    CFF_RETURN_LOCAL:
        IF NOT bReturnEntryBlocked THEN
            IF bReturnPublicationAllowed THEN
                IF bStateEntry THEN
                    udiZCommandId := udiZCommandId + 1;
                    IF udiZCommandId = 0 THEN
                        udiZCommandId := 1;
                    END_IF
                END_IF
                stMotionIntent.stZCommand.bEnable := TRUE;
                stMotionIntent.stZCommand.bReset := FALSE;
                stMotionIntent.stZCommand.bStop := FALSE;
                stMotionIntent.stZCommand.bHome := FALSE;
                stMotionIntent.stZCommand.bMoveAbsolute := TRUE;
                stMotionIntent.stZCommand.bMoveVelocity := FALSE;
                stMotionIntent.stZCommand.bUseExternalSetpoint := FALSE;
                stMotionIntent.stZCommand.rHomePosition_mm := 0.0;
                stMotionIntent.stZCommand.rPosition_mm := rCycleStartZPosition_mm;
                stMotionIntent.stZCommand.rVelocity_mm_s :=
                    stCycleSnapshot.stProgram.stHeader.fReturnVelocityMmS;
                stMotionIntent.stZCommand.rAcceleration_mm_s2 :=
                    stSequenceConfigSnapshot.fStandardMoveAccelerationMmS2;
                stMotionIntent.stZCommand.rDeceleration_mm_s2 :=
                    stSequenceConfigSnapshot.fStandardMoveDecelerationMmS2;
                stMotionIntent.stZCommand.eOwnerRequest := Z_OWNER_RETRACT;
                stMotionIntent.bExternalEnableRequest := FALSE;
                stMotionIntent.bExternalDisableRequest := FALSE;
                stMotionIntent.rExternalTargetVelocity_mm_s := 0.0;
                stMotionIntent.bForceProcessExitComplete := TRUE;
                stMotionIntent.bRAxisProcessRequested := TRUE;
                stMotionIntent.stRCommand.bEnable := TRUE;
                stMotionIntent.stRCommand.bReset := FALSE;
                stMotionIntent.stRCommand.bStop := TRUE;
                stMotionIntent.stRCommand.bMoveVelocity := FALSE;
                stMotionIntent.stRCommand.rVelocity_rpm := 0.0;
                stMotionIntent.stRCommand.rAcceleration_rpm_s :=
                    stRAxisProfileSnapshot.fSpeedRampRpmS;
                stMotionIntent.stRCommand.rDeceleration_rpm_s :=
                    stRAxisProfileSnapshot.fSpeedRampRpmS;
                bForceControlEnable := FALSE;
                IF tonReturn.Q THEN
                    IF udiFirstFaultId = 0 THEN
                        udiFirstFaultId := 16#0000A015;
                    END_IF
                    eExitIntent := CFF_EXIT_FAULT_NO_RETURN;
                    eNextState := CFF_FAULT;
                END_IF
                IF (GVL_Status.stFast.udiAcceptedSequenceZCommandId = udiZCommandId)
                    AND GVL_Status.stFast.stZAxis.bDone
                    AND GVL_Status.stFast.stZAxis.bStandstill
                    AND NOT tonReturn.Q THEN
                    eNextState := CFF_EVALUATE;
                END_IF
            ELSE
                IF udiFirstFaultId = 0 THEN
                    udiFirstFaultId := 16#0000A016;
                END_IF
                eExitIntent := CFF_EXIT_FAULT_NO_RETURN;
                eNextState := CFF_FAULT;
            END_IF
        END_IF
    CFF_RETURN_REFERENCE:
        IF NOT bReturnEntryBlocked THEN
            IF bReturnPublicationAllowed THEN
                IF bStateEntry THEN
                    udiZCommandId := udiZCommandId + 1;
                    IF udiZCommandId = 0 THEN
                        udiZCommandId := 1;
                    END_IF
                END_IF
                stMotionIntent.stZCommand.bEnable := TRUE;
                stMotionIntent.stZCommand.bReset := FALSE;
                stMotionIntent.stZCommand.bStop := FALSE;
                stMotionIntent.stZCommand.bHome := FALSE;
                stMotionIntent.stZCommand.bMoveAbsolute := TRUE;
                stMotionIntent.stZCommand.bMoveVelocity := FALSE;
                stMotionIntent.stZCommand.bUseExternalSetpoint := FALSE;
                stMotionIntent.stZCommand.rHomePosition_mm := 0.0;
                stMotionIntent.stZCommand.rPosition_mm :=
                    stCycleSnapshot.stProgram.stHeader.fReturnOpeningMm;
                stMotionIntent.stZCommand.rVelocity_mm_s :=
                    stCycleSnapshot.stProgram.stHeader.fReturnVelocityMmS;
                stMotionIntent.stZCommand.rAcceleration_mm_s2 :=
                    stSequenceConfigSnapshot.fStandardMoveAccelerationMmS2;
                stMotionIntent.stZCommand.rDeceleration_mm_s2 :=
                    stSequenceConfigSnapshot.fStandardMoveDecelerationMmS2;
                stMotionIntent.stZCommand.eOwnerRequest := Z_OWNER_RETRACT;
                stMotionIntent.bExternalEnableRequest := FALSE;
                stMotionIntent.bExternalDisableRequest := FALSE;
                stMotionIntent.rExternalTargetVelocity_mm_s := 0.0;
                stMotionIntent.bForceProcessExitComplete := TRUE;
                stMotionIntent.bRAxisProcessRequested := TRUE;
                stMotionIntent.stRCommand.bEnable := TRUE;
                stMotionIntent.stRCommand.bReset := FALSE;
                stMotionIntent.stRCommand.bStop := TRUE;
                stMotionIntent.stRCommand.bMoveVelocity := FALSE;
                stMotionIntent.stRCommand.rVelocity_rpm := 0.0;
                stMotionIntent.stRCommand.rAcceleration_rpm_s :=
                    stRAxisProfileSnapshot.fSpeedRampRpmS;
                stMotionIntent.stRCommand.rDeceleration_rpm_s :=
                    stRAxisProfileSnapshot.fSpeedRampRpmS;
                bForceControlEnable := FALSE;
                IF tonReturn.Q THEN
                    IF udiFirstFaultId = 0 THEN
                        udiFirstFaultId := 16#0000A015;
                    END_IF
                    eExitIntent := CFF_EXIT_FAULT_NO_RETURN;
                    eNextState := CFF_FAULT;
                END_IF
                IF (GVL_Status.stFast.udiAcceptedSequenceZCommandId = udiZCommandId)
                    AND GVL_Status.stFast.stZAxis.bDone
                    AND GVL_Status.stFast.stZAxis.bStandstill
                    AND NOT tonReturn.Q THEN
                    eNextState := CFF_EVALUATE;
                END_IF
            ELSE
                IF udiFirstFaultId = 0 THEN
                    udiFirstFaultId := 16#0000A016;
                END_IF
                eExitIntent := CFF_EXIT_FAULT_NO_RETURN;
                eNextState := CFF_FAULT;
            END_IF
        END_IF
    CFF_EVALUATE:
        stMotionIntent.stZCommand.bEnable := TRUE;
        stMotionIntent.stZCommand.bReset := FALSE;
        stMotionIntent.stZCommand.bStop := FALSE;
        stMotionIntent.stZCommand.bHome := FALSE;
        stMotionIntent.stZCommand.bMoveAbsolute := TRUE;
        stMotionIntent.stZCommand.bMoveVelocity := FALSE;
        stMotionIntent.stZCommand.bUseExternalSetpoint := FALSE;
        stMotionIntent.stZCommand.rHomePosition_mm := 0.0;
        stMotionIntent.stZCommand.rPosition_mm := SEL(
            stCycleSnapshot.stProgram.stHeader.eReturnMode = RETURN_MODE_REFERENCE,
            rCycleStartZPosition_mm,
            stCycleSnapshot.stProgram.stHeader.fReturnOpeningMm);
        stMotionIntent.stZCommand.rVelocity_mm_s :=
            stCycleSnapshot.stProgram.stHeader.fReturnVelocityMmS;
        stMotionIntent.stZCommand.rAcceleration_mm_s2 :=
            stSequenceConfigSnapshot.fStandardMoveAccelerationMmS2;
        stMotionIntent.stZCommand.rDeceleration_mm_s2 :=
            stSequenceConfigSnapshot.fStandardMoveDecelerationMmS2;
        stMotionIntent.stZCommand.eOwnerRequest := Z_OWNER_RETRACT;
        stMotionIntent.bExternalEnableRequest := FALSE;
        stMotionIntent.bExternalDisableRequest := FALSE;
        stMotionIntent.rExternalTargetVelocity_mm_s := 0.0;
        stMotionIntent.bForceProcessExitComplete := TRUE;
        stMotionIntent.bRAxisProcessRequested := TRUE;
        stMotionIntent.stRCommand.bEnable := TRUE;
        stMotionIntent.stRCommand.bReset := FALSE;
        stMotionIntent.stRCommand.bStop := TRUE;
        stMotionIntent.stRCommand.bMoveVelocity := FALSE;
        stMotionIntent.stRCommand.rVelocity_rpm := 0.0;
        stMotionIntent.stRCommand.rAcceleration_rpm_s := stRAxisProfileSnapshot.fSpeedRampRpmS;
        stMotionIntent.stRCommand.rDeceleration_rpm_s := stRAxisProfileSnapshot.fSpeedRampRpmS;
        bForceControlEnable := FALSE;
        nWrittenStepPrefix := 0;
        bStepResultHole := FALSE;
        bMissingStepResult := FALSE;
        bEvaluateNok := FALSE;
        bEvaluateFault := FALSE;
        FOR nStepIndex := 1 TO 4 DO
            IF abStepResultWritten[nStepIndex] THEN
                IF NOT bMissingStepResult THEN
                    nWrittenStepPrefix := nStepIndex;
                END_IF
                IF bMissingStepResult THEN
                    bStepResultHole := TRUE;
                END_IF
                bEvaluateNok := bEvaluateNok
                    OR GVL_Process.astStepCriterion[nStepIndex].bNok
                    OR GVL_Process.astStepCriterion[nStepIndex].bTooShort
                    OR GVL_Process.astStepCriterion[nStepIndex].bSecondaryLatched
                    OR (GVL_Process.astStepCriterion[nStepIndex].eEndCause
                        = STEP_END_MAX_TIME);
            ELSE
                bMissingStepResult := TRUE;
            END_IF
        END_FOR
        IF abStepResultWritten[4] THEN
            bEvaluateNok := bEvaluateNok
                OR NOT GVL_Process.astStepCriterion[4].bQualifiedForceHoldMet;
        END_IF
        bEvaluateFault := bStepResultHole;
        IF eExitIntent = CFF_EXIT_NORMAL_RETURN THEN
            IF (nWrittenStepPrefix <> 4) OR bEvaluateNok THEN
                bEvaluateFault := TRUE;
            END_IF
        ELSIF eExitIntent = CFF_EXIT_NOK_RETURN THEN
            IF NOT ((nWrittenStepPrefix >= 1) AND bEvaluateNok) THEN
                bEvaluateFault := TRUE;
            END_IF
        ELSIF eExitIntent = CFF_EXIT_ABORT_NO_RETURN THEN
            bEvaluateFault := FALSE;
        ELSE
            bEvaluateFault := TRUE;
        END_IF
        IF bEvaluateFault THEN
            IF udiFirstFaultId = 0 THEN
                udiFirstFaultId := 16#0000A016;
            END_IF
            eExitIntent := CFF_EXIT_FAULT_NO_RETURN;
        END_IF
        IF (eExitIntent = CFF_EXIT_NORMAL_RETURN) AND NOT bEvaluateFault THEN
            eNextState := CFF_COMPLETE_OK;
        ELSIF (eExitIntent = CFF_EXIT_NOK_RETURN) AND NOT bEvaluateFault THEN
            eNextState := CFF_COMPLETE_NOK;
        ELSIF (eExitIntent = CFF_EXIT_ABORT_NO_RETURN) AND NOT bEvaluateFault THEN
            eNextState := CFF_ABORT;
        ELSE
            eNextState := CFF_FAULT;
        END_IF
    CFF_COMPLETE_OK:
        stMotionIntent.stZCommand.bEnable := TRUE;
        stMotionIntent.stZCommand.bReset := FALSE;
        stMotionIntent.stZCommand.bStop := FALSE;
        stMotionIntent.stZCommand.bHome := FALSE;
        stMotionIntent.stZCommand.bMoveAbsolute := TRUE;
        stMotionIntent.stZCommand.bMoveVelocity := FALSE;
        stMotionIntent.stZCommand.bUseExternalSetpoint := FALSE;
        stMotionIntent.stZCommand.rHomePosition_mm := 0.0;
        stMotionIntent.stZCommand.rPosition_mm := SEL(
            stCycleSnapshot.stProgram.stHeader.eReturnMode = RETURN_MODE_REFERENCE,
            rCycleStartZPosition_mm,
            stCycleSnapshot.stProgram.stHeader.fReturnOpeningMm);
        stMotionIntent.stZCommand.rVelocity_mm_s :=
            stCycleSnapshot.stProgram.stHeader.fReturnVelocityMmS;
        stMotionIntent.stZCommand.rAcceleration_mm_s2 :=
            stSequenceConfigSnapshot.fStandardMoveAccelerationMmS2;
        stMotionIntent.stZCommand.rDeceleration_mm_s2 :=
            stSequenceConfigSnapshot.fStandardMoveDecelerationMmS2;
        stMotionIntent.stZCommand.eOwnerRequest := Z_OWNER_RETRACT;
        stMotionIntent.bExternalEnableRequest := FALSE;
        stMotionIntent.bExternalDisableRequest := FALSE;
        stMotionIntent.rExternalTargetVelocity_mm_s := 0.0;
        stMotionIntent.bForceProcessExitComplete := TRUE;
        stMotionIntent.bRAxisProcessRequested := TRUE;
        stMotionIntent.stRCommand.bEnable := TRUE;
        stMotionIntent.stRCommand.bReset := FALSE;
        stMotionIntent.stRCommand.bStop := TRUE;
        stMotionIntent.stRCommand.bMoveVelocity := FALSE;
        stMotionIntent.stRCommand.rVelocity_rpm := 0.0;
        stMotionIntent.stRCommand.rAcceleration_rpm_s := stRAxisProfileSnapshot.fSpeedRampRpmS;
        stMotionIntent.stRCommand.rDeceleration_rpm_s := stRAxisProfileSnapshot.fSpeedRampRpmS;
        bForceControlEnable := FALSE;
        IF GVL_Status.stFast.stZAxis.bStandstill
            AND GVL_Status.stFast.stRAxis.bStandstill
            AND bExternalReady THEN
            bBusy := FALSE;
            bDone := TRUE;
            bError := FALSE;
            bAborted := FALSE;
        END_IF
    CFF_COMPLETE_NOK:
        stMotionIntent.stZCommand.bEnable := TRUE;
        stMotionIntent.stZCommand.bReset := FALSE;
        stMotionIntent.stZCommand.bStop := FALSE;
        stMotionIntent.stZCommand.bHome := FALSE;
        stMotionIntent.stZCommand.bMoveAbsolute := TRUE;
        stMotionIntent.stZCommand.bMoveVelocity := FALSE;
        stMotionIntent.stZCommand.bUseExternalSetpoint := FALSE;
        stMotionIntent.stZCommand.rHomePosition_mm := 0.0;
        stMotionIntent.stZCommand.rPosition_mm := SEL(
            stCycleSnapshot.stProgram.stHeader.eReturnMode = RETURN_MODE_REFERENCE,
            rCycleStartZPosition_mm,
            stCycleSnapshot.stProgram.stHeader.fReturnOpeningMm);
        stMotionIntent.stZCommand.rVelocity_mm_s :=
            stCycleSnapshot.stProgram.stHeader.fReturnVelocityMmS;
        stMotionIntent.stZCommand.rAcceleration_mm_s2 :=
            stSequenceConfigSnapshot.fStandardMoveAccelerationMmS2;
        stMotionIntent.stZCommand.rDeceleration_mm_s2 :=
            stSequenceConfigSnapshot.fStandardMoveDecelerationMmS2;
        stMotionIntent.stZCommand.eOwnerRequest := Z_OWNER_RETRACT;
        stMotionIntent.bExternalEnableRequest := FALSE;
        stMotionIntent.bExternalDisableRequest := FALSE;
        stMotionIntent.rExternalTargetVelocity_mm_s := 0.0;
        stMotionIntent.bForceProcessExitComplete := TRUE;
        stMotionIntent.bRAxisProcessRequested := TRUE;
        stMotionIntent.stRCommand.bEnable := TRUE;
        stMotionIntent.stRCommand.bReset := FALSE;
        stMotionIntent.stRCommand.bStop := TRUE;
        stMotionIntent.stRCommand.bMoveVelocity := FALSE;
        stMotionIntent.stRCommand.rVelocity_rpm := 0.0;
        stMotionIntent.stRCommand.rAcceleration_rpm_s := stRAxisProfileSnapshot.fSpeedRampRpmS;
        stMotionIntent.stRCommand.rDeceleration_rpm_s := stRAxisProfileSnapshot.fSpeedRampRpmS;
        bForceControlEnable := FALSE;
        IF GVL_Status.stFast.stZAxis.bStandstill
            AND GVL_Status.stFast.stRAxis.bStandstill
            AND bExternalReady THEN
            bBusy := FALSE;
            bDone := TRUE;
            bError := TRUE;
            bAborted := FALSE;
        END_IF
    CFF_ABORT:
        IF bStateEntry AND bTerminalFaultStopRequired
            AND NOT bApproachFaultStopPending THEN
            udiZCommandId := udiZCommandId + 1;
            IF udiZCommandId = 0 THEN
                udiZCommandId := 1;
            END_IF
            bApproachFaultStopPending := TRUE;
            bTerminalFaultStopRequired := FALSE;
        END_IF
        stMotionIntent.stZCommand.bEnable := TRUE;
        stMotionIntent.stZCommand.bReset := FALSE;
        stMotionIntent.stZCommand.bStop := TRUE;
        stMotionIntent.stZCommand.bHome := FALSE;
        stMotionIntent.stZCommand.bMoveAbsolute := FALSE;
        stMotionIntent.stZCommand.bMoveVelocity := FALSE;
        stMotionIntent.stZCommand.bUseExternalSetpoint := FALSE;
        stMotionIntent.stZCommand.rHomePosition_mm := 0.0;
        stMotionIntent.stZCommand.rPosition_mm := 0.0;
        stMotionIntent.stZCommand.rVelocity_mm_s := 0.0;
        stMotionIntent.stZCommand.rAcceleration_mm_s2 := stSequenceConfigSnapshot.fStandardMoveAccelerationMmS2;
        stMotionIntent.stZCommand.rDeceleration_mm_s2 := stSequenceConfigSnapshot.fStandardMoveDecelerationMmS2;
        stMotionIntent.stZCommand.eOwnerRequest := Z_OWNER_FAULT_STOP;
        stMotionIntent.bExternalEnableRequest := FALSE;
        stMotionIntent.bExternalDisableRequest := FALSE;
        stMotionIntent.rExternalTargetVelocity_mm_s := 0.0;
        stMotionIntent.bForceProcessExitComplete := TRUE;
        stMotionIntent.bRAxisProcessRequested := TRUE;
        stMotionIntent.stRCommand.bEnable := TRUE;
        stMotionIntent.stRCommand.bReset := FALSE;
        stMotionIntent.stRCommand.bStop := TRUE;
        stMotionIntent.stRCommand.bMoveVelocity := FALSE;
        stMotionIntent.stRCommand.rVelocity_rpm := 0.0;
        stMotionIntent.stRCommand.rAcceleration_rpm_s := stRAxisProfileSnapshot.fSpeedRampRpmS;
        stMotionIntent.stRCommand.rDeceleration_rpm_s := stRAxisProfileSnapshot.fSpeedRampRpmS;
        bForceControlEnable := FALSE;
        IF bApproachFaultStopPending
            AND (GVL_Status.stFast.udiAcceptedSequenceZCommandId = udiZCommandId)
            AND GVL_Status.stFast.stZAxis.bStandstill
            AND (GVL_Status.stFast.udiAcceptedSequenceRCommandId = udiRCommandId)
            AND GVL_Status.stFast.stRAxis.bStandstill THEN
            bApproachFaultStopPending := FALSE;
        END_IF
        IF NOT bApproachFaultStopPending
            AND GVL_Status.stFast.stZAxis.bStandstill
            AND GVL_Status.stFast.stRAxis.bStandstill
            AND bExternalReady THEN
            bBusy := FALSE;
            bDone := FALSE;
            bError := FALSE;
            bAborted := TRUE;
        END_IF
    CFF_FAULT:
        IF udiFirstFaultId = 0 THEN
            udiFirstFaultId := 16#0000A016;
        END_IF
        IF bStateEntry AND bTerminalFaultStopRequired
            AND NOT bApproachFaultStopPending THEN
            udiZCommandId := udiZCommandId + 1;
            IF udiZCommandId = 0 THEN
                udiZCommandId := 1;
            END_IF
            bApproachFaultStopPending := TRUE;
            bTerminalFaultStopRequired := FALSE;
        END_IF
        stMotionIntent.stZCommand.bEnable := TRUE;
        stMotionIntent.stZCommand.bReset := FALSE;
        stMotionIntent.stZCommand.bStop := TRUE;
        stMotionIntent.stZCommand.bHome := FALSE;
        stMotionIntent.stZCommand.bMoveAbsolute := FALSE;
        stMotionIntent.stZCommand.bMoveVelocity := FALSE;
        stMotionIntent.stZCommand.bUseExternalSetpoint := FALSE;
        stMotionIntent.stZCommand.rHomePosition_mm := 0.0;
        stMotionIntent.stZCommand.rPosition_mm := 0.0;
        stMotionIntent.stZCommand.rVelocity_mm_s := 0.0;
        stMotionIntent.stZCommand.rAcceleration_mm_s2 := stSequenceConfigSnapshot.fStandardMoveAccelerationMmS2;
        stMotionIntent.stZCommand.rDeceleration_mm_s2 := stSequenceConfigSnapshot.fStandardMoveDecelerationMmS2;
        stMotionIntent.stZCommand.eOwnerRequest := Z_OWNER_FAULT_STOP;
        stMotionIntent.bExternalEnableRequest := FALSE;
        stMotionIntent.bExternalDisableRequest := FALSE;
        stMotionIntent.rExternalTargetVelocity_mm_s := 0.0;
        stMotionIntent.bForceProcessExitComplete := TRUE;
        stMotionIntent.bRAxisProcessRequested := TRUE;
        stMotionIntent.stRCommand.bEnable := TRUE;
        stMotionIntent.stRCommand.bReset := FALSE;
        stMotionIntent.stRCommand.bStop := TRUE;
        stMotionIntent.stRCommand.bMoveVelocity := FALSE;
        stMotionIntent.stRCommand.rVelocity_rpm := 0.0;
        stMotionIntent.stRCommand.rAcceleration_rpm_s := stRAxisProfileSnapshot.fSpeedRampRpmS;
        stMotionIntent.stRCommand.rDeceleration_rpm_s := stRAxisProfileSnapshot.fSpeedRampRpmS;
        bForceControlEnable := FALSE;
        IF bApproachFaultStopPending
            AND (GVL_Status.stFast.udiAcceptedSequenceZCommandId = udiZCommandId)
            AND GVL_Status.stFast.stZAxis.bStandstill
            AND (GVL_Status.stFast.udiAcceptedSequenceRCommandId = udiRCommandId)
            AND GVL_Status.stFast.stRAxis.bStandstill THEN
            bApproachFaultStopPending := FALSE;
        END_IF
        IF NOT bApproachFaultStopPending
            AND GVL_Status.stFast.stZAxis.bStandstill
            AND GVL_Status.stFast.stRAxis.bStandstill
            AND bExternalReady THEN
            bBusy := FALSE;
            bDone := FALSE;
            bError := TRUE;
            bAborted := FALSE;
        END_IF
ELSE
    IF udiFirstFaultId = 0 THEN
        udiFirstFaultId := 16#0000A016;
    END_IF
    eExitIntent := CFF_EXIT_FAULT_NO_RETURN;
    IF NOT bExternalReady THEN
        (* Unknown state while External still owns the axis: preserve the
           active Z identity/owner contract and create a fresh R stop. *)
        IF udiZCommandId = 0 THEN
            udiZCommandId := 1;
        END_IF
        udiRCommandId := udiRCommandId + 1;
        IF udiRCommandId = 0 THEN
            udiRCommandId := 1;
        END_IF
        bUnknownExternalRStopPending := TRUE;
        stMotionIntent.stZCommand.bEnable := TRUE;
        stMotionIntent.stZCommand.bReset := FALSE;
        stMotionIntent.stZCommand.bStop := FALSE;
        stMotionIntent.stZCommand.bHome := FALSE;
        stMotionIntent.stZCommand.bMoveAbsolute := FALSE;
        stMotionIntent.stZCommand.bMoveVelocity := FALSE;
        stMotionIntent.stZCommand.eOwnerRequest := Z_OWNER_FORCE_PROCESS;
        stMotionIntent.stZCommand.bUseExternalSetpoint := TRUE;
        stMotionIntent.stZCommand.rHomePosition_mm := 0.0;
        stMotionIntent.stZCommand.rPosition_mm := 0.0;
        stMotionIntent.stZCommand.rVelocity_mm_s := 0.0;
        stMotionIntent.stZCommand.rAcceleration_mm_s2 := 0.0;
        stMotionIntent.stZCommand.rDeceleration_mm_s2 :=
            stSequenceConfigSnapshot.fStandardMoveDecelerationMmS2;
        stMotionIntent.bExternalEnableRequest := FALSE;
        stMotionIntent.bExternalDisableRequest := TRUE;
        stMotionIntent.rExternalTargetVelocity_mm_s := 0.0;
        stMotionIntent.bForceProcessExitComplete := FALSE;
        stMotionIntent.bRAxisProcessRequested := TRUE;
        stMotionIntent.stRCommand.bEnable := TRUE;
        stMotionIntent.stRCommand.bReset := FALSE;
        stMotionIntent.stRCommand.bStop := TRUE;
        stMotionIntent.stRCommand.bMoveVelocity := FALSE;
        stMotionIntent.stRCommand.rVelocity_rpm := 0.0;
        stMotionIntent.stRCommand.rAcceleration_rpm_s := stRAxisProfileSnapshot.fSpeedRampRpmS;
        stMotionIntent.stRCommand.rDeceleration_rpm_s := stRAxisProfileSnapshot.fSpeedRampRpmS;
        bForceControlEnable := FALSE;
        eNextState := CFF_EXTSETPOINT_DISABLE;
    ELSE
        (* External is released, so terminate any possible standard NC motion
           with one fresh FaultStop transaction and retain the R zero-stop. *)
        udiZCommandId := udiZCommandId + 1;
        IF udiZCommandId = 0 THEN
            udiZCommandId := 1;
        END_IF
        udiRCommandId := udiRCommandId + 1;
        IF udiRCommandId = 0 THEN
            udiRCommandId := 1;
        END_IF
        bApproachFaultStopPending := TRUE;
        stMotionIntent.stZCommand.bEnable := TRUE;
        stMotionIntent.stZCommand.bReset := FALSE;
        stMotionIntent.stZCommand.bStop := TRUE;
        stMotionIntent.stZCommand.bHome := FALSE;
        stMotionIntent.stZCommand.bMoveAbsolute := FALSE;
        stMotionIntent.stZCommand.bMoveVelocity := FALSE;
        stMotionIntent.stZCommand.eOwnerRequest := Z_OWNER_FAULT_STOP;
        stMotionIntent.stZCommand.bUseExternalSetpoint := FALSE;
        stMotionIntent.stZCommand.rHomePosition_mm := 0.0;
        stMotionIntent.stZCommand.rPosition_mm := 0.0;
        stMotionIntent.stZCommand.rVelocity_mm_s := 0.0;
        stMotionIntent.stZCommand.rAcceleration_mm_s2 := stSequenceConfigSnapshot.fStandardMoveAccelerationMmS2;
        stMotionIntent.stZCommand.rDeceleration_mm_s2 := stSequenceConfigSnapshot.fStandardMoveDecelerationMmS2;
        stMotionIntent.bExternalEnableRequest := FALSE;
        stMotionIntent.bExternalDisableRequest := FALSE;
        stMotionIntent.rExternalTargetVelocity_mm_s := 0.0;
        stMotionIntent.bRAxisProcessRequested := TRUE;
        stMotionIntent.stRCommand.bEnable := TRUE;
        stMotionIntent.stRCommand.bReset := FALSE;
        stMotionIntent.stRCommand.bStop := TRUE;
        stMotionIntent.stRCommand.bMoveVelocity := FALSE;
        stMotionIntent.stRCommand.rVelocity_rpm := 0.0;
        stMotionIntent.stRCommand.rAcceleration_rpm_s := stRAxisProfileSnapshot.fSpeedRampRpmS;
        stMotionIntent.stRCommand.rDeceleration_rpm_s := stRAxisProfileSnapshot.fSpeedRampRpmS;
        bForceControlEnable := FALSE;
        eNextState := CFF_FAULT;
    END_IF
END_CASE

(* 唯一结果发布点：先构造完整payload，再写公开槽位，最后锁存guard。 *)
IF bStepResultPublishRequested AND NOT abStepResultWritten[nStepResultIndex] THEN
    stStepResultCandidate := stClearedStepCriterionResult;
    stStepResultCandidate.eStep := eStep;
    stStepResultCandidate.eEndCause := fbStepCriterion.stOutput.eEndCause;
    stStepResultCandidate.bPrimaryLatched := fbStepCriterion.stOutput.bPrimaryMet;
    stStepResultCandidate.bSecondaryLatched :=
        fbStepCriterion.stOutput.bSecondaryLimitReached;
    stStepResultCandidate.bNok := bStepResultNok;
    stStepResultCandidate.nTriggerCycle := GVL_Status.stFast.nCycleCounter;
    stStepResultCandidate.bTooShort := fbStepCriterion.stOutput.bTooShort;
    stStepResultCandidate.bQualifiedForceHoldMet := (nStepResultIndex = 4)
        AND (uliQualifiedHold_us >= uliQualifiedHoldTarget_us);
    stStepResultCandidate.rQualifiedForceHoldTime_s := rQualifiedForceHoldTime_s;
    stStepResultCandidate.rLatchedForce_kN :=
        fbStepCriterion.stOutput.rLatchedForce_kN;
    stStepResultCandidate.rLatchedRelativePosition_mm :=
        fbStepCriterion.stOutput.rLatchedRelativePosition_mm;
    stStepResultCandidate.rLatchedStepTime_s :=
        fbStepCriterion.stOutput.rLatchedStepTime_s;
    GVL_Process.astStepCriterion[nStepResultIndex] := stStepResultCandidate;
    abStepResultWritten[nStepResultIndex] := TRUE;
END_IF

(* This classifier is evaluated after the state branch so a newly latched
   timeout/algorithm fault is routed to safety in the same Fast scan. *)
bSafeExitRequested := bStopRequestedLatched OR bAbortEvent OR bResetPendingLatched
    OR bHardForceActive OR bHardStrokeActive OR bCollisionLimitActive
    OR bExternalError OR bAxisError OR bSensorInvalid OR (udiFirstFaultId > 0);
bReturnSafeStopRequested := ((eState = CFF_RETURN_LOCAL)
        OR (eState = CFF_RETURN_REFERENCE)
        OR (eState = CFF_EVALUATE)
        OR (eState = CFF_COMPLETE_OK)
        OR (eState = CFF_COMPLETE_NOK))
    AND bSafeExitRequested;

(* Return-capable intent never survives a same-scan real fault or active event. *)
IF (udiFirstFaultId > 0) OR bHardForceActive OR bHardStrokeActive
    OR bCollisionLimitActive OR bExternalError OR bAxisError OR bSensorInvalid THEN
    eExitIntent := CFF_EXIT_FAULT_NO_RETURN;
ELSIF bStopRequestedLatched OR bAbortEvent OR bResetPendingLatched THEN
    eExitIntent := CFF_EXIT_ABORT_NO_RETURN;
END_IF

(* Disable may have selected Abort before a same-scan real fault was normalized. *)
IF (eState = CFF_EXTSETPOINT_DISABLE)
    AND (eNextState = CFF_ABORT)
    AND (eExitIntent = CFF_EXIT_FAULT_NO_RETURN) THEN
    eNextState := CFF_FAULT;
END_IF

(* Abort等待中出现的真实故障必须覆盖Abort，但不改写已锁存的更早首故障。 *)
IF (eState = CFF_ABORT) AND (eExitIntent = CFF_EXIT_FAULT_NO_RETURN) THEN
    eNextState := CFF_FAULT;
END_IF

(* A same-scan hard/error/abort path cannot withdraw the External owner before release. *)
IF bExternalOwnerHold AND bSafeExitRequested THEN
    stMotionIntent.stZCommand.bEnable := TRUE;
    stMotionIntent.stZCommand.eOwnerRequest := Z_OWNER_FORCE_PROCESS;
    stMotionIntent.stZCommand.bUseExternalSetpoint := TRUE;
    stMotionIntent.rExternalTargetVelocity_mm_s := 0.0;
    stMotionIntent.bForceProcessExitComplete := FALSE;
    stMotionIntent.bRAxisProcessRequested := TRUE;
    stCandidateRCommand.bEnable := TRUE;
    stCandidateRCommand.bReset := FALSE;
    stCandidateRCommand.bStop := TRUE;
    stCandidateRCommand.bMoveVelocity := FALSE;
    stCandidateRCommand.rVelocity_rpm := 0.0;
    stCandidateRCommand.rAcceleration_rpm_s := stRAxisProfileSnapshot.fSpeedRampRpmS;
    stCandidateRCommand.rDeceleration_rpm_s := stRAxisProfileSnapshot.fSpeedRampRpmS;
    stMotionIntent.stRCommand := stCandidateRCommand;
    bSafeExitRStopPending := TRUE;
    IF stCandidateRCommand.bEnable <> stLastPublishedRCommand.bEnable
        OR stCandidateRCommand.bReset <> stLastPublishedRCommand.bReset
        OR stCandidateRCommand.bStop <> stLastPublishedRCommand.bStop
        OR stCandidateRCommand.bMoveVelocity <> stLastPublishedRCommand.bMoveVelocity
        OR stCandidateRCommand.rVelocity_rpm <> stLastPublishedRCommand.rVelocity_rpm
        OR stCandidateRCommand.rAcceleration_rpm_s
            <> stLastPublishedRCommand.rAcceleration_rpm_s
        OR stCandidateRCommand.rDeceleration_rpm_s
            <> stLastPublishedRCommand.rDeceleration_rpm_s THEN
        stLastPublishedRCommand := stCandidateRCommand;
        stMotionIntent.stRCommand := stCandidateRCommand;
        udiRCommandId := udiRCommandId + 1;
        IF udiRCommandId = 0 THEN
            udiRCommandId := 1;
        END_IF
    END_IF
    bForceControlEnable := FALSE;
    IF (eExitIntent = CFF_EXIT_ABORT_NO_RETURN)
        AND bUnloadHealthy
        AND (eState >= CFF_CONTACT_SEARCH)
        AND (eState <= CFF_CONTROLLED_FORCE_UNLOAD) THEN
        stMotionIntent.bExternalEnableRequest := TRUE;
        stMotionIntent.bExternalDisableRequest := FALSE;
        bForceControlEnable := TRUE;
        rForceSet_kN := 0.0;
        IF eState < CFF_CONTROLLED_FORCE_UNLOAD THEN
            IF NOT bUnloadTransferInitialized THEN
                rTargetRelativePosition_mm := GVL_Process.stActual.fSRelSensorMm;
                rForceTransferVelocity_mm_s :=
                    GVL_Status.stFast.stZExtSetpoint.rAcceptedVelocity_mm_s;
                bForceProfileTransferPending := TRUE;
                bUnloadTransferInitialized := TRUE;
            END_IF
            eNextState := CFF_CONTROLLED_FORCE_UNLOAD;
        END_IF
    ELSE
        stMotionIntent.bExternalEnableRequest := FALSE;
        stMotionIntent.bExternalDisableRequest := TRUE;
        bForceControlEnable := FALSE;
        eNextState := CFF_EXTSETPOINT_DISABLE;
    END_IF
END_IF

(* If release and a safety cause arrive in the same scan, the state branch may
   already have rebuilt an Enable request.  The strictly positive release gate
   therefore overrides the complete payload with fresh standard stop identities. *)
IF GVL_Status.stFast.stZExtSetpoint.bReleaseOwner THEN
    IF bExternalProcessState
        AND GVL_Status.stFast.stZExtSetpoint.bReleaseOwner
        AND bSafeExitRequested THEN
        udiZCommandId := udiZCommandId + 1;
        IF udiZCommandId = 0 THEN
            udiZCommandId := 1;
        END_IF
        udiRCommandId := udiRCommandId + 1;
        IF udiRCommandId = 0 THEN
            udiRCommandId := 1;
        END_IF
        bApproachFaultStopPending := TRUE;
        stMotionIntent.bExternalEnableRequest := FALSE;
        stMotionIntent.bExternalDisableRequest := FALSE;
        stMotionIntent.rExternalTargetVelocity_mm_s := 0.0;
        stMotionIntent.bForceProcessExitComplete := TRUE;
        stMotionIntent.stZCommand.bEnable := TRUE;
        stMotionIntent.stZCommand.bReset := FALSE;
        stMotionIntent.stZCommand.bStop := TRUE;
        stMotionIntent.stZCommand.bHome := FALSE;
        stMotionIntent.stZCommand.bMoveAbsolute := FALSE;
        stMotionIntent.stZCommand.bMoveVelocity := FALSE;
        stMotionIntent.stZCommand.eOwnerRequest := Z_OWNER_FAULT_STOP;
        stMotionIntent.stZCommand.bUseExternalSetpoint := FALSE;
        stMotionIntent.stZCommand.rHomePosition_mm := 0.0;
        stMotionIntent.stZCommand.rPosition_mm := 0.0;
        stMotionIntent.stZCommand.rVelocity_mm_s := 0.0;
        stMotionIntent.stZCommand.rAcceleration_mm_s2 := stSequenceConfigSnapshot.fStandardMoveAccelerationMmS2;
        stMotionIntent.stZCommand.rDeceleration_mm_s2 := stSequenceConfigSnapshot.fStandardMoveDecelerationMmS2;
        stMotionIntent.bRAxisProcessRequested := TRUE;
        stMotionIntent.stRCommand.bEnable := TRUE;
        stMotionIntent.stRCommand.bReset := FALSE;
        stMotionIntent.stRCommand.bStop := TRUE;
        stMotionIntent.stRCommand.bMoveVelocity := FALSE;
        stMotionIntent.stRCommand.rVelocity_rpm := 0.0;
        stMotionIntent.stRCommand.rAcceleration_rpm_s := stRAxisProfileSnapshot.fSpeedRampRpmS;
        stMotionIntent.stRCommand.rDeceleration_rpm_s := stRAxisProfileSnapshot.fSpeedRampRpmS;
        bForceControlEnable := FALSE;
        IF eExitIntent = CFF_EXIT_ABORT_NO_RETURN THEN
            eNextState := CFF_ABORT;
        ELSE
            eExitIntent := CFF_EXIT_FAULT_NO_RETURN;
            eNextState := CFF_FAULT;
        END_IF
    END_IF
END_IF

(* Return/Evaluate/Complete的同扫安全事件在状态分支之后覆盖Done，并只创建一次FaultStop事务。 *)
IF bReturnSafeStopRequested THEN
    IF NOT bApproachFaultStopPending THEN
        udiZCommandId := udiZCommandId + 1;
        IF udiZCommandId = 0 THEN
            udiZCommandId := 1;
        END_IF
        bApproachFaultStopPending := TRUE;
    END_IF
    stMotionIntent.stZCommand.bEnable := TRUE;
    stMotionIntent.stZCommand.bReset := FALSE;
    stMotionIntent.stZCommand.bStop := TRUE;
    stMotionIntent.stZCommand.bHome := FALSE;
    stMotionIntent.stZCommand.bMoveAbsolute := FALSE;
    stMotionIntent.stZCommand.bMoveVelocity := FALSE;
    stMotionIntent.stZCommand.bUseExternalSetpoint := FALSE;
    stMotionIntent.stZCommand.rHomePosition_mm := 0.0;
    stMotionIntent.stZCommand.rPosition_mm := 0.0;
    stMotionIntent.stZCommand.rVelocity_mm_s := 0.0;
    stMotionIntent.stZCommand.rAcceleration_mm_s2 :=
        stSequenceConfigSnapshot.fStandardMoveAccelerationMmS2;
    stMotionIntent.stZCommand.rDeceleration_mm_s2 :=
        stSequenceConfigSnapshot.fStandardMoveDecelerationMmS2;
    stMotionIntent.stZCommand.eOwnerRequest := Z_OWNER_FAULT_STOP;
    stMotionIntent.bExternalEnableRequest := FALSE;
    stMotionIntent.bExternalDisableRequest := FALSE;
    stMotionIntent.rExternalTargetVelocity_mm_s := 0.0;
    stMotionIntent.bForceProcessExitComplete := TRUE;
    stMotionIntent.bRAxisProcessRequested := TRUE;
    stMotionIntent.stRCommand.bEnable := TRUE;
    stMotionIntent.stRCommand.bReset := FALSE;
    stMotionIntent.stRCommand.bStop := TRUE;
    stMotionIntent.stRCommand.bMoveVelocity := FALSE;
    stMotionIntent.stRCommand.rVelocity_rpm := 0.0;
    stMotionIntent.stRCommand.rAcceleration_rpm_s := stRAxisProfileSnapshot.fSpeedRampRpmS;
    stMotionIntent.stRCommand.rDeceleration_rpm_s := stRAxisProfileSnapshot.fSpeedRampRpmS;
    bForceControlEnable := FALSE;
    IF eExitIntent = CFF_EXIT_FAULT_NO_RETURN THEN
        eNextState := CFF_FAULT;
    ELSE
        eExitIntent := CFF_EXIT_ABORT_NO_RETURN;
        eNextState := CFF_ABORT;
    END_IF
END_IF

(* Precheck owns no motion, so active Stop/Abort/Reset can route directly to a
   terminal wait without depending on the asynchronous Contact Reset ACK. *)
IF eState = CFF_PRECHECK AND bPrecheckExitRequested THEN
    IF eExitIntent = CFF_EXIT_ABORT_NO_RETURN THEN
        eNextState := CFF_ABORT;
    ELSE
        eExitIntent := CFF_EXIT_FAULT_NO_RETURN;
        eNextState := CFF_FAULT;
    END_IF
END_IF

(* Approach has not entered External and may use the standard Fault Stop path. *)
IF eState = CFF_APPROACH AND bSafeExitRequested THEN
    IF NOT bApproachFaultStopPending THEN
        udiZCommandId := udiZCommandId + 1;
        IF udiZCommandId = 0 THEN
            udiZCommandId := 1;
        END_IF
        bApproachFaultStopPending := TRUE;
    END_IF
    stMotionIntent.stZCommand.bEnable := TRUE;
    stMotionIntent.stZCommand.bReset := FALSE;
    stMotionIntent.stZCommand.bStop := TRUE;
    stMotionIntent.stZCommand.bHome := FALSE;
    stMotionIntent.stZCommand.bMoveAbsolute := FALSE;
    stMotionIntent.stZCommand.bMoveVelocity := FALSE;
    stMotionIntent.stZCommand.eOwnerRequest := Z_OWNER_FAULT_STOP;
    stMotionIntent.stZCommand.bUseExternalSetpoint := FALSE;
    stMotionIntent.stZCommand.rHomePosition_mm := 0.0;
    stMotionIntent.stZCommand.rPosition_mm := 0.0;
    stMotionIntent.stZCommand.rVelocity_mm_s := 0.0;
    stMotionIntent.stZCommand.rAcceleration_mm_s2 := stSequenceConfigSnapshot.fStandardMoveAccelerationMmS2;
    stMotionIntent.stZCommand.rDeceleration_mm_s2 := stSequenceConfigSnapshot.fStandardMoveDecelerationMmS2;
    stMotionIntent.bExternalDisableRequest := FALSE;
    IF tonRAxisStop.Q
        OR (udiFirstFaultId = 16#0000A014) THEN
        eExitIntent := CFF_EXIT_FAULT_NO_RETURN;
        eNextState := CFF_FAULT;
    ELSIF tonApproach.Q THEN
        IF udiFirstFaultId = 0 THEN
            udiFirstFaultId := 16#0000A007;
        END_IF
        eExitIntent := CFF_EXIT_FAULT_NO_RETURN;
        eNextState := CFF_FAULT;
    ELSIF (GVL_Status.stFast.udiAcceptedSequenceZCommandId = udiZCommandId)
        AND GVL_Status.stFast.stZAxis.bStandstill
        AND (GVL_Status.stFast.udiAcceptedSequenceRCommandId = udiRCommandId)
        AND GVL_Status.stFast.stRAxis.bStandstill THEN
        bApproachFaultStopPending := FALSE;
        IF eExitIntent = CFF_EXIT_ABORT_NO_RETURN THEN
            eNextState := CFF_ABORT;
        ELSIF eExitIntent = CFF_EXIT_FAULT_NO_RETURN THEN
            eNextState := CFF_FAULT;
        ELSE
            IF udiFirstFaultId = 0 THEN
                udiFirstFaultId := 16#0000A016;
            END_IF
            eExitIntent := CFF_EXIT_FAULT_NO_RETURN;
            eNextState := CFF_FAULT;
        END_IF
    ELSE
        eNextState := eState;
    END_IF
END_IF

IF (eState = CFF_IDLE) AND NOT bSafeTerminalReset
    AND (bStopRequestedLatched OR bAbortEvent OR bResetPendingLatched) THEN
    eExitIntent := CFF_EXIT_ABORT_NO_RETURN;
    eNextState := CFF_ABORT;
END_IF

IF (eState = CFF_IDLE) AND (udiFirstFaultId <> 0) THEN
    bBusy := TRUE;
    eExitIntent := CFF_EXIT_FAULT_NO_RETURN;
    eNextState := CFF_FAULT;
END_IF

(* Contact publisher: five payload fields first and the RequestId last, at one site only. *)
IF bProcessReferencePending THEN
    GVL_Command.stProcessReference.bLatchContactReference :=
        stPendingProcessReferenceCommand.bLatchContactReference;
    GVL_Command.stProcessReference.bUseProvidedContactReference :=
        stPendingProcessReferenceCommand.bUseProvidedContactReference;
    GVL_Command.stProcessReference.rProvidedContactSensorPosition_mm :=
        stPendingProcessReferenceCommand.rProvidedContactSensorPosition_mm;
    GVL_Command.stProcessReference.rProvidedContactAxisPosition_mm :=
        stPendingProcessReferenceCommand.rProvidedContactAxisPosition_mm;
    GVL_Command.stProcessReference.bResetContactReference :=
        stPendingProcessReferenceCommand.bResetContactReference;
    GVL_Command.stProcessReference.udiContactReferenceRequestId :=
        stPendingProcessReferenceCommand.udiContactReferenceRequestId;
END_IF

(* A profile-transfer request is retained until Force is actually enabled. *)
IF bForceProfileTransferPending AND bForceControlEnable THEN
    bForceProfileTransfer := TRUE;
    bForceProfileTransferPending := FALSE;
END_IF

IF bSafeTerminalReset THEN
    bBusy := FALSE;
    bDone := FALSE;
    bError := FALSE;
    bAborted := FALSE;
    bStopRequestedLatched := FALSE;
    bResetPendingLatched := FALSE;
    bCycleNokLatched := FALSE;
    udiFirstFaultId :=0;
    udiActiveStartCommandId := 0;
    bStartSourceSnapshotConsistent := FALSE;
    eExitIntent := CFF_EXIT_NONE;
    eStep := CFF_STEP_NONE;
    eSubPhase := STEP_SUBPHASE_NONE;
    eEndCause := STEP_END_NONE;
    stFastConfigSnapshot.bValid := FALSE;
    bForceControlEnable := FALSE;
    bForceProfileTransfer := FALSE;
    bForceProfileTransferPending := FALSE;
    rForceTransferVelocity_mm_s := 0.0;
    rForceSet_kN := 0.0;
    rForceRamp_kN_s := 0.0;
    rSpeedSet_rpm := 0.0;
    rTargetRelativePosition_mm := 0.0;
    rHardMaximumRelativePosition_mm := 0.0;
    rRequiredRelativePosition_mm := 0.0;
    rStepBoundary_mm := 0.0;
    rCycleStartZPosition_mm := 0.0;
    rStepTime_s := 0.0;
    rQualifiedForceHoldTime_s := 0.0;
    uliCycleDelta_us := 0;
    uliStepElapsed_us := 0;
    uliStepMaximum_us := 0;
    uliQualifiedHold_us := 0;
    uliQualifiedHoldTarget_us := 0;
    bRpmStopped := FALSE;
    bForceInBand := FALSE;
    bStepResultPublishRequested := FALSE;
    bStepResultNok := FALSE;
    nStepResultIndex := 1;
    bEvaluateNok := FALSE;
    bEvaluateFault := FALSE;
    bStepResultHole := FALSE;
    bMissingStepResult := FALSE;
    nWrittenStepPrefix := 0;
    bHardForceActive := FALSE;
    bHardStrokeActive := FALSE;
    bCollisionLimitActive := FALSE;
    bProcessReferencePending := FALSE;
    bProcessReferenceResetPending := FALSE;
    bProcessReferenceLatchPending := FALSE;
    bApproachFaultStopPending := FALSE;
    bUnknownExternalRStopPending := FALSE;
    bSafeExitRStopPending := FALSE;
    bTerminalFaultStopRequired := FALSE;
    bUnloadTransferInitialized := FALSE;
    bContactResetPulse := TRUE;
    bForceDeclineResetPulse := TRUE;
    bStepCriterionResetPulse := TRUE;
    eNextState := CFF_IDLE;
END_IF

(* Stop is the final diagnostic end cause until Start or safe Reset clears it. *)
IF bStopRequestedLatched THEN
    eEndCause := STEP_END_STOP_REQUEST;
END_IF

(* A transition scan never publishes the completed truth table of its source state. *)
IF (eState <> eNextState)
    AND ((eNextState = CFF_ABORT) OR (eNextState = CFF_FAULT)) THEN
    bBusy := TRUE;
    bDone := FALSE;
    bError := FALSE;
    bAborted := FALSE;
END_IF

(* Publish stable source identities and the complete typed Sequence status. *)
stMotionIntent.udiZCommandId := udiZCommandId;
stMotionIntent.udiRCommandId := udiRCommandId;
GVL_Status.stFast.stSequence.nAcceptedCommandId := udiActiveStartCommandId;
GVL_Status.stFast.stSequence.bBusy := bBusy;
GVL_Status.stFast.stSequence.bDone := bDone;
GVL_Status.stFast.stSequence.bAborted := bAborted;
GVL_Status.stFast.stSequence.bError := bError;
GVL_Status.stFast.stSequence.nErrorId := udiFirstFaultId;
GVL_Status.stFast.stSequence.eState := eNextState;
GVL_Status.stFast.stSequence.eStep := eStep;
GVL_Status.stFast.stSequence.eSubPhase := eSubPhase;
GVL_Status.stFast.stSequence.eEndCause := eEndCause;
GVL_Status.stFast.stSequence.eExitIntent := eExitIntent;
GVL_Status.stFast.stSequence.bCycleNok := bCycleNokLatched;
GVL_Status.stFast.stSequence.bRpmStopped := bRpmStopped;
GVL_Status.stFast.stSequence.bForceInBand := bForceInBand;
GVL_Status.stFast.stSequence.rStepTime_s := rStepTime_s;
GVL_Status.stFast.stSequence.rQualifiedForceHoldTime_s := rQualifiedForceHoldTime_s;
GVL_Status.stFast.stSequence.rForceSet_kN := rForceSet_kN;
GVL_Status.stFast.stSequence.rForceRamp_kN_s := rForceRamp_kN_s;
GVL_Status.stFast.stSequence.bForceControlEnable := bForceControlEnable;
GVL_Status.stFast.stSequence.bForceProfileTransfer := bForceProfileTransfer;
GVL_Status.stFast.stSequence.rForceTransferVelocity_mm_s := rForceTransferVelocity_mm_s;
GVL_Status.stFast.stSequence.rTargetRelativePosition_mm := rTargetRelativePosition_mm;
GVL_Status.stFast.stSequence.rHardMaximumRelativePosition_mm := rHardMaximumRelativePosition_mm;
GVL_Status.stFast.stSequence.bForceHardLimitActive := bHardForceActive;
GVL_Status.stFast.stSequence.bStrokeHardLimitActive := bHardStrokeActive;
GVL_Status.stFast.stSequence.bCollisionLimitActive := bCollisionLimitActive;
GVL_Status.stFast.stSequence.rSpeedSet_rpm := rSpeedSet_rpm;
GVL_Status.stFast.stSequence.stContact := fbContactDetect.stOutput;
GVL_Status.stFast.stSequence.stForceDecline := fbForceDecline.stOutput;
GVL_Status.stFast.stSequence.stStepCriterion := fbStepCriterion.stOutput;
GVL_Status.stFast.stSequence.stMotionIntent := stMotionIntent;
GVL_Status.stFast.stSequence.stFastConfigSnapshot := stFastConfigSnapshot;

GVL_Alarm.astRequests[9].eCode := E_AlarmCode.ALARM_CFF_CRITERION_FAULT;
GVL_Alarm.astRequests[9].eLevel := E_AlarmLevel.ALARM_LEVEL_FAULT;
GVL_Alarm.astRequests[9].nTextId := 3000;
GVL_Alarm.astRequests[9].nSourceId := 9;
GVL_Alarm.astRequests[9].bLatch := TRUE;
GVL_Alarm.astRequests[9].bActive := fbContactDetect.stOutput.bFault
    OR fbForceDecline.stOutput.bFault
    OR fbStepCriterion.stOutput.bFault;
GVL_Alarm.astRequests[10].eCode := E_AlarmCode.ALARM_CFF_SEQUENCE_FAULT;
GVL_Alarm.astRequests[10].eLevel := E_AlarmLevel.ALARM_LEVEL_FAULT;
GVL_Alarm.astRequests[10].nTextId := 3200;
GVL_Alarm.astRequests[10].nSourceId := 10;
GVL_Alarm.astRequests[10].bLatch := TRUE;
GVL_Alarm.astRequests[10].bActive := udiFirstFaultId <> 0;

(* Exactly one state assignment completes the scan. *)
ePreviousState := eState;
eState := eNextState;
bStateEntry := eState <> ePreviousState;

END_PROGRAM

(* stored: Version 1.1.0.1
   POU PRG_CffSequence: Id {A2000000-0000-4000-8000-000000000002} *)
